Fanuc KAREL source: ADD_BYNAMEPC.kl

PROGRAM T
%NOLOCKGROUP
VAR
 v0 : ARRAY[20] OF BYTE
 v1 : INTEGER
 v2 : STRING[40]
 v3 : STRING[40]
 v4 : INTEGER
BEGIN
 ADD_BYNAMEPC(v0, v1, v2, v3, v4)
END T
